PROGRAM LadderMain
VAR_IN_OUT //from MAIN
	removeBundleLeft : BOOL;
	removeBundleRight : BOOL;
END_VAR
VAR_OUTPUT
	bundleIn : Bundle;
	bundleOut : Bundle;
	
	ready : BOOL;
	busy : BOOL;
	done : BOOL;
	
	error : BOOL;
	backlog : BOOL;
	
	localTime : TIMESTRUCT;
	pause : BOOL;
END_VAR
VAR
	setup : BOOL;
	
	retrievedTcpData : AdsData;
	
	expectedBundles : ARRAY[0..GVL.maxQueue] OF STRING; //bundles expected to arrive
	expectedArrivals : ARRAY[0..GVL.maxQueue] OF TIMESTRUCT; //bundles expected to arrive
	numEtaBundles : INT;
	
	newBundle : POINTER TO Bundle; //arrived bundle for A2.6
	newBypass : POINTER TO BOOL;
	
	inputBundle : POINTER TO Bundle; //input buffer
	
	//spacerRecollector : PackagerFreeAsync; //:= (sectionId := 6); //spacer recollector section
	//packagingSection : PackagerFreeAsync; //packaging section
	
	paperSection : PaperEx;
	cardboardCornerGuardSection : CardboardCornerGuardEx;
	chipboardSection : ChipboardEx;
	woodBunkSection : WoodBunkEx;
	outputSection : AreaOutputEx;
	
	runPaper : BOOL := TRUE;
	runCardboardCornerGuard : BOOL := TRUE;
	runChipboard : BOOL := TRUE;
	runWoodBunk : BOOL := TRUE;
	runOutput : BOOL := TRUE;
		
	outputBuffer : ARRAY[Surface.LEFT..Surface.RIGHT] OF POINTER TO Bundle; //output buffer
	numOutputBundles : USINT := 0;
	
	fbLocalSystemTime : FB_LocalSystemTime;
END_VAR
VAR CONSTANT
	maxOutputBundles : USINT := 3;
END_VAR
VAR // added by the converter: edge detectors and wires of the graphical bodies
    _w1 : BOOL;
END_VAR

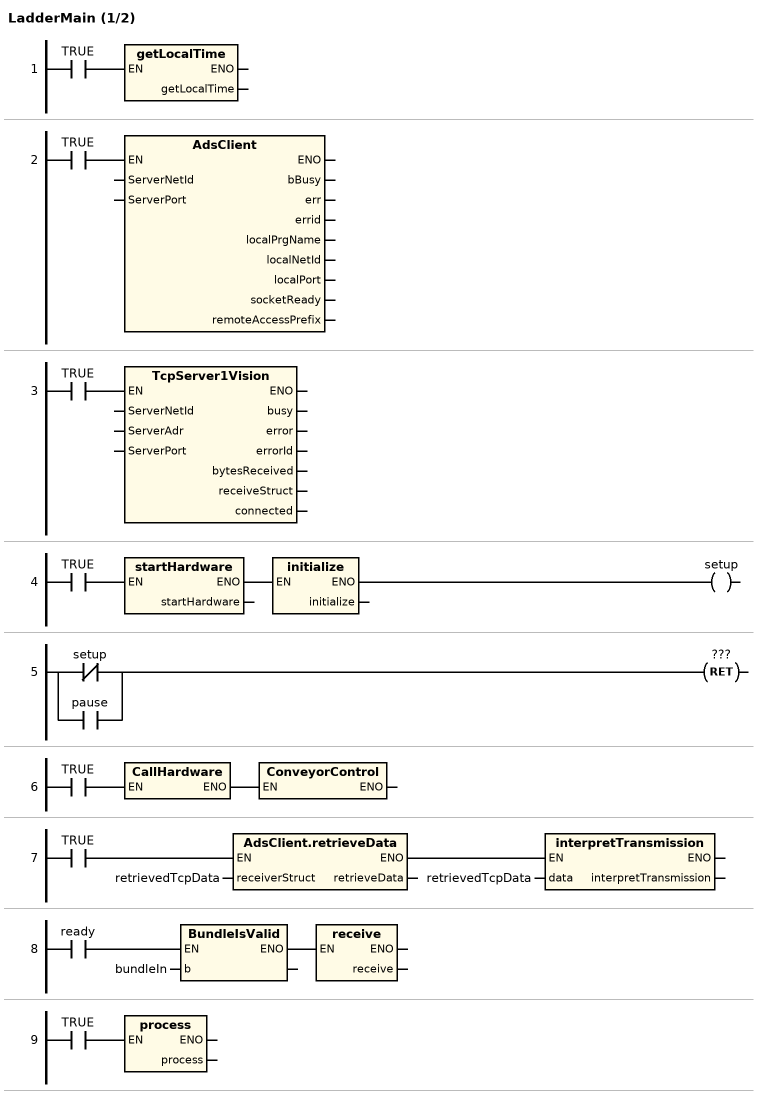
// NETWORK 1
getLocalTime();

// NETWORK 2
AdsClient();

// NETWORK 3
TcpServer1Vision();

// NETWORK 4
startHardware();
initialize();
setup := TRUE;

// NETWORK 5
IF NOT setup OR pause THEN RETURN; END_IF

// NETWORK 6
CallHardware();
ConveyorControl();

// NETWORK 7
AdsClient.retrieveData(receiverStruct := retrievedTcpData);
interpretTransmission(data := retrievedTcpData);

// NETWORK 8
_w1 := ready;
IF _w1 THEN BundleIsValid(b := bundleIn); END_IF
IF _w1 THEN receive(); END_IF

// NETWORK 9
process();

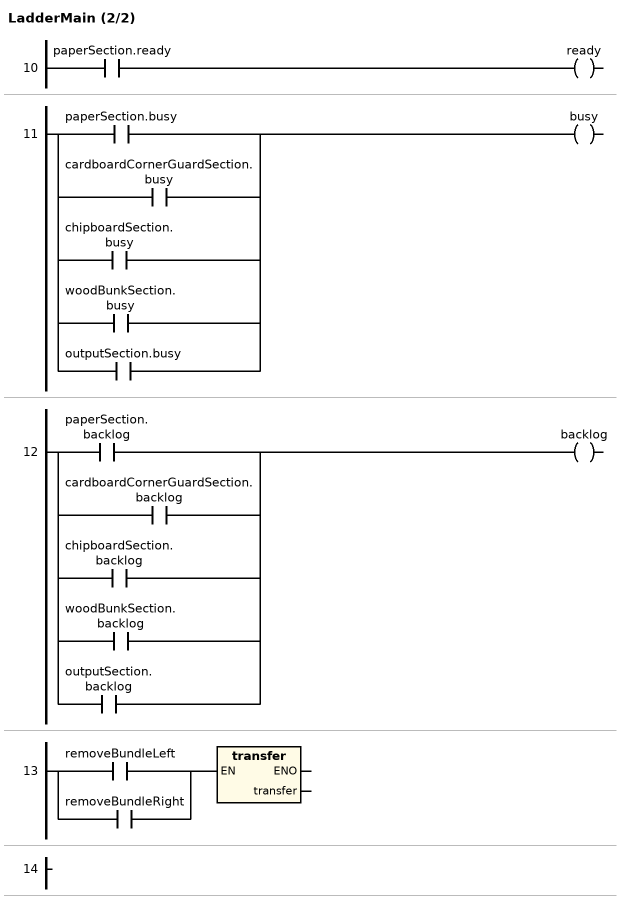
// NETWORK 10
ready := paperSection.ready;

// NETWORK 11
busy := paperSection.busy OR cardboardCornerGuardSection.busy OR chipboardSection.busy OR woodBunkSection.busy OR outputSection.busy;

// NETWORK 12
backlog := paperSection.backlog OR cardboardCornerGuardSection.backlog OR chipboardSection.backlog OR woodBunkSection.backlog OR outputSection.backlog;

// NETWORK 13
IF removeBundleLeft OR removeBundleRight THEN transfer(); END_IF

// NETWORK 14

METHOD PRIVATE complete : BOOL //tcpip read
//area 2 is an end of line, send bundles to buffer and log in local + system database
(*
(*
temp := outputBundles.pop();

GVL.bundlesCompleted.push(value := temp^.id);
GVL.events.push(value := EventsEnum.AREA_COMPLETE);

__DELETE(temp); //deallocate memory of bundle leaving A2.5

//log and signal back to dispatch PLC
GVL.events.push(value := EventsEnum.AREA_COMPLETE);
*)

IF numOutputBundles < maxOutputBundles THEN //if output has space, move to output and start next bundle
	MEMCPY(ADR(outputBundles[numOutputBundles]), packagingSection.bundleOut, SIZEOF(Bundle));
	__DELETE(packagingSection.bundleOut);
	
	//run conveyor until bundle is in output buffer
	packagingSection.resetStatus();
	
	done := TRUE; //mark PLC as done for Dispatch to acknowledge
END_IF
//do nothing if output center is occupied

(*
IF NOT BundleIsValid(GVL.bundleOut) THEN //bundle was removed from output buffer
	MEMMOVE(ADR(outputBundles[0]), ADR(outputBundles[1]), SIZEOF(outputBundles) - SIZEOF(outputBundles[0]));
	outputBundles[maxOutputBundles-1] := nullBundle;
	
	GVL.bundleOut := outputBundles[0];
	
	numOutputBundles := numOutputBundles - 1;
END_IF
*)
*)
END_METHOD

METHOD PRIVATE getLocalTime : BOOL
VAR_INPUT
END_VAR
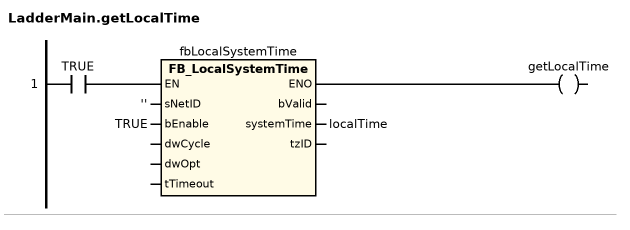
// NETWORK 1
fbLocalSystemTime(sNetID := '', bEnable := TRUE, systemTime => localTime); // FB_LocalSystemTime
getLocalTime := TRUE;
END_METHOD

METHOD PRIVATE initialize : BOOL
(*
prepare the program data types
*)
paperSection.connectTo(ADR(cardboardCornerGuardSection));
cardboardCornerGuardSection.connectTo(ADR(chipboardSection));
chipboardSection.connectTo(ADR(woodBunkSection));
woodBunkSection.connectTo(ADR(outputSection));

(*
12, 20	entry + paper
9, 11	cardboard + corner guard
5, 8	chipboard + wood bunk
1, 4 	output buffer

0, 0 	spacer recollector (possibly obsolete)
*)
paperSection.assignConveyors(12, 20);
cardboardCornerGuardSection.assignConveyors(9, 11);
chipboardSection.assignConveyors(5, 8);
woodBunkSection.assignConveyors(5, 8);
outputSection.assignConveyors(1, 4);

initialize := TRUE;
END_METHOD

METHOD PRIVATE interpretTransmission : BOOL
VAR_INPUT
	data : REFERENCE TO AdsData;
END_VAR
VAR
	i : INT;
END_VAR
CASE data.description OF
	EventsEnum.BUNDLE_IN:
		MEMCPY(ADR(bundleIn), ADR(data.binaryData), SIZEOF(bundleIn));
			
	EventsEnum.BUNDLE_ETA:
		MEMCPY(ADR(expectedBundles[numEtaBundles]), ADR(data.binaryData), SIZEOF(expectedBundles[numEtaBundles]));
		expectedArrivals[numEtaBundles] := data.timestamp;
		
END_CASE
END_METHOD

METHOD PRIVATE process : BOOL
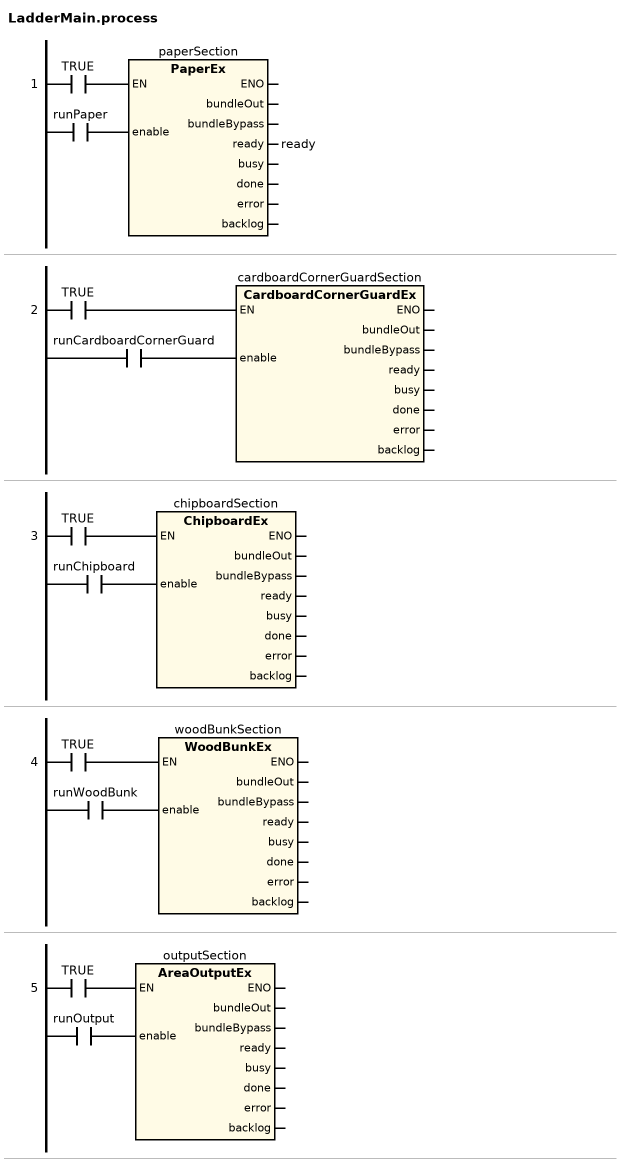
// NETWORK 1
paperSection(enable := runPaper, ready => ready); // PaperEx

// NETWORK 2
cardboardCornerGuardSection(enable := runCardboardCornerGuard); // CardboardCornerGuardEx

// NETWORK 3
chipboardSection(enable := runChipboard); // ChipboardEx

// NETWORK 4
woodBunkSection(enable := runWoodBunk); // WoodBunkEx

// NETWORK 5
outputSection(enable := runOutput); // AreaOutputEx
END_METHOD

METHOD PRIVATE receive : BOOL
VAR
	i : INT;
	shiftIndex : INT := -1;
	invalidBundle : Bundle;
END_VAR
(*
1 - find bundle in bundle ETAs and remove
2 - add bundle to all sections' queues and reset bundle
*)
ready := FALSE;
busy := TRUE;
done := FALSE;

FOR i:=0 TO GVL.maxQueue BY 1 DO
	IF expectedBundles[i] = bundleIn.id THEN
		shiftIndex := i;
		EXIT;
	END_IF
END_FOR

IF shiftIndex > -1 THEN //shift everything down
	MEMMOVE(
		ADR(expectedBundles[shiftIndex]), 
		ADR(expectedBundles[shiftIndex + 1]), 
		SIZEOF(STRING) * TO_UINT(GVL.maxQueue - shiftIndex));
		
	MEMMOVE(
		ADR(expectedArrivals[shiftIndex]), 
		ADR(expectedArrivals[shiftIndex + 1]), 
		SIZEOF(TIMESTRUCT) * TO_UINT(GVL.maxQueue - shiftIndex) );
		
	numEtaBundles := numEtaBundles - 1;
END_IF


newBundle := __NEW(Bundle);
newBundle^ := bundleIn;

newBypass := __NEW(BOOL);
newBypass^ := FALSE;

paperSection.queueBundle(newBundle, newBypass);
cardboardCornerGuardSection.queueBundle(newBundle, newBypass);
chipboardSection.queueBundle(newBundle, newBypass);
woodBunkSection.queueBundle(newBundle, newBypass);
outputSection.queueBundle(newBundle, newBypass);

bundleIn := invalidBundle; //reset bundle
END_METHOD

METHOD PRIVATE startHardware : BOOL
END_METHOD

METHOD PRIVATE transfer : BOOL
VAR
	i : INT;
END_VAR
//send TCP/ADS transmission back to Dispatch once bundle is removed from the plant
(*
FOR i:=Surface.LEFT TO Surface.RIGHT BY 1 DO
	

	IF removeBundle[i] AND outputBuffer[i] <> 0 THEN
		//log data
		__DELETE(outputBuffer[i]);
	END_IF


END_FOR
*)
END_METHOD

END_PROGRAM

(* stored: Version 1.1.0.1, ProductVersion 3.1.4024.11
   POU LadderMain: Id {7843ca70-049b-4185-a9be-f6a0bd1c14ed}, SpecialFunc None
   Method complete: Id {0c34d03b-4d96-4815-aa03-24ed7b7fda1c}
   Method getLocalTime: Id {d1e96e49-69b2-4ce5-a264-7e537a235e11}
   Method initialize: Id {208b5a5c-ae00-4394-8a4d-6652b6fa171a}
   Method interpretTransmission: Id {c31d12ae-0a38-4d84-980a-d258289b6031}
   Method process: Id {a26908e1-f81b-43f6-b5cf-376e1d437673}
   Method receive: Id {9a10cbb4-f21d-4089-949e-dd412777be9d}
   Method startHardware: Id {ceb42471-ed88-41cb-8de8-1b541926b427}
   Method transfer: Id {8065d680-2ec5-4670-b0a5-f998499670ad} *)
